INTERFACE I_List EXTENDS I_Collection

METHOD PUBLIC GetIndexOf : DINT
VAR_INPUT
	Item : ANY;
END_VAR
END_METHOD

METHOD Insert : BOOL
VAR_INPUT
	Index : DINT;
	Item : ANY;
END_VAR
END_METHOD

METHOD PUBLIC Item : I_ListNode
VAR_INPUT
	Index : DINT;
END_VAR
END_METHOD

METHOD RemoveAt : BOOL
VAR_INPUT
	Index : DINT;
END_VAR
END_METHOD

END_INTERFACE

(* stored: Version 1.1.0.1, ProductVersion 3.1.4024.12
   Itf I_List: Id {412a2b67-91e4-4aae-a3d3-321ed0ca4b34}
   Method GetIndexOf: Id {d91cdb09-c4a3-48f7-934b-f0ebbd93f0cb}
   Method Insert: Id {61d79cd2-a37c-4e6b-96ef-c3dcdf52a503}
   Method Item: Id {f4065bfd-8f7c-416b-935b-6682e135dc7d}
   Method RemoveAt: Id {3fd904de-394f-4ea8-8de5-3698783696e0} *)
